Staubli VAL3: Control_PanelS.pgx

public program Control_PanelS(string x_sTitle, num x_nLTopX, num x_nLTopY, num x_nWidthX, num x_nLengthY)
  local num l_nIndex
begin
  //画有标题的框



  //设定框的位置与大小
  call Control_PanelXY(x_nLTopX,x_nLTopY,x_nWidthX,x_nLengthY)

  //文本显示状况进行设定
   call Control_Panel(x_sTitle)









end
